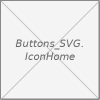
VISUALIZATION ButtonHome  // 100x100
VAR_IN_OUT
	bState : BOOL;
END_VAR
    Frame (0,0 100x100)
        shows ButtonTemplate(bActive := bState)
    Image (0,0 100x100), image: Buttons_SVG.IconHome
        OnMouseDown: execute { GVL_HMI.fbHMIControl.eScreenRequest := E_BaseVisu.Idle; }
END_VISUALIZATION

(* stored: Version 1.1.0.1, ProductVersion 3.1.4024.11
   Visu ButtonHome: Id {f774b592-26be-4399-a0be-9d92794926b9} *)
